INTERFACE ITF_UdpConnection EXTENDS ITF_Cyclic

METHOD IsConnected : BOOL
VAR_INPUT
END_VAR
END_METHOD

METHOD IsSending : BOOL
VAR_INPUT
END_VAR
END_METHOD

PROPERTY ReceiveBufferReference : REFERENCE TO ARRAY [0..TCPADS_MAXUDP_BUFFSIZE - 1] OF BYTE;
GET
END_GET
END_PROPERTY

METHOD TryCloseConnection : HRESULT
VAR_INPUT
END_VAR
END_METHOD

METHOD TryOpenConnection : HRESULT
VAR_INPUT
END_VAR
END_METHOD

METHOD TrySendData : HRESULT
VAR_INPUT
	IpAddress		: T_IPv4Addr;
	Port			: UDINT;
	DataAddress		: PVOID;
	DataLength		: UDINT;
END_VAR
END_METHOD

END_INTERFACE

(* stored: Version 1.1.0.1
   Itf ITF_UdpConnection: Id {94303b2c-fab7-40fd-a3af-21426bd39a97}
   Method IsConnected: Id {7d024eb6-e212-4edc-bc9d-ebb6925af72c}
   Method IsSending: Id {4a057512-f722-4737-be05-87be5a8c18a8}
   Property ReceiveBufferReference: Id {c42e4fae-ab30-4073-bdff-c9d721aed2a4}
   Get Get: Id {d15e6cd2-50b2-4e14-ae3f-231b8211d661}
   Method TryCloseConnection: Id {23fdee8e-f6c9-4523-af56-7d00a02774a6}
   Method TryOpenConnection: Id {1124eedc-b83d-4b70-a9f5-afd5bd113767}
   Method TrySendData: Id {6796c252-d973-40c6-9a54-4cbc36b15f3b} *)
